// TIA Portal V19 export
DATA_BLOCK "NEW INPUTS"   // DB68
{ S7_Optimized_Access := 'TRUE' }
// stored: MemoryReserve 100
   VAR
      "EMG STOP IP" : Bool;
      "PHASE FAIL IP" : Bool;
      "HOOTER RESET IP" : Bool;
      "HOOTER RESET HMI" : Bool;
      "AUTO/MAN SW IP" : Bool;
      "MGF FEED PUMP RUN IP" : Bool;
      "RO 1 HPP RUN IP" : Bool;
      "RO 2 HPP RUN IP" : Bool;
      "CIP PUMP RUN IP" : Bool;
      "PW TRANSFER PUMP - W RUN IP" : Bool;
      "PW TRANSFER PUMP - S RUN IP" : Bool;
      "PW TRANSFER W/P" : Bool;
      "AIR PRESSURE FAIL" : Bool;
      "SPARE IP3" : Bool;
      "LS-5 TANK LOW IP" : Bool;
      "LS-5 TANK HIGH IP" : Bool;
      "SPARE IP4" : Bool;
      "SPARE IP5" : Bool;
      "SPARE IP6" : Bool;
      "SPARE IP7" : Bool;
      "SPARE IP8" : Bool;
      "LPS-1" : Bool;
      "LPS-2" : Bool;
      "MGF V-1 OPEN FB" : Bool;
      "MGF V-2 OPEN FB" : Bool;
      "MGF V-3 OPEN FB" : Bool;
      "MGF V-4 OPEN FB" : Bool;
      "MGF V-1 CLOSE FB" : Bool;
      "MGF V-2 CLOSE FB" : Bool;
      "MGF V-3 CLOSE FB" : Bool;
      "MGF V-4 CLOSE FB" : Bool;
      "MGF V-5 OPEN FB" : Bool;
      "MGF V-5 CLOSE FB" : Bool;
      "ACF OPEN FB V1" : Bool;
      "ACF OPEN FB V2" : Bool;
      "ACF OPEN FB V3" : Bool;
      "ACF OPEN FB V4" : Bool;
      "ACF OPEN FB V5" : Bool;
      "ACF CLOSE FB V1" : Bool;
      "ACF CLOSE FB V2" : Bool;
      "ACF CLOSE FB V3" : Bool;
      "ACF CLOSE FB V4" : Bool;
      "ACF CLOSE FB V5" : Bool;
      "SF OPEN FB V1" : Bool;
      "SF OPEN FB V2" : Bool;
      "SF OPEN FB V3" : Bool;
      "SF OPEN FB V4" : Bool;
      "SF OPEN FB V5" : Bool;
      "SF OPEN FB V6" : Bool;
      "SF OPEN FB V7" : Bool;
      "SF CLOSE FB V1" : Bool;
      "SF CLOSE FB V2" : Bool;
      "SF CLOSE FB V3" : Bool;
      "SF CLOSE FB V4" : Bool;
      "SF CLOSE FB V5" : Bool;
      "SF CLOSE FB V6" : Bool;
      "SF CLOSE FB V7" : Bool;
      "SPARE IP9" : Bool;
      "SPARE IP10" : Bool;
      "SPARE IP11" : Bool;
      "SPARE IP12" : Bool;
      "SPARE IP13" : Bool;
      "SPARE IP14" : Bool;
   END_VAR
BEGIN
END_DATA_BLOCK
